% RSLogix 500 project PLC_Level_2_Project_9.RSS, saved by version 8.30.00.16 %
PROJECT "UNTITLED"    % processor: Bul.1763 MicroLogix 1100 Series B %

PROGRAM FILES
  LAD 2   8 rungs

DATA FILES
  O0 OUTPUT  4 elements
  I1 INPUT  6 elements
  S2 STATUS  66 elements
  B3 BINARY  1 elements
  T4 TIMER  1 elements
  C5 COUNTER  1 elements
  R6 CONTROL  1 elements
  N7 INTEGER  4 elements
  F8 FLOAT  1 elements
  ST9 STRING  8 elements

LADDER 2
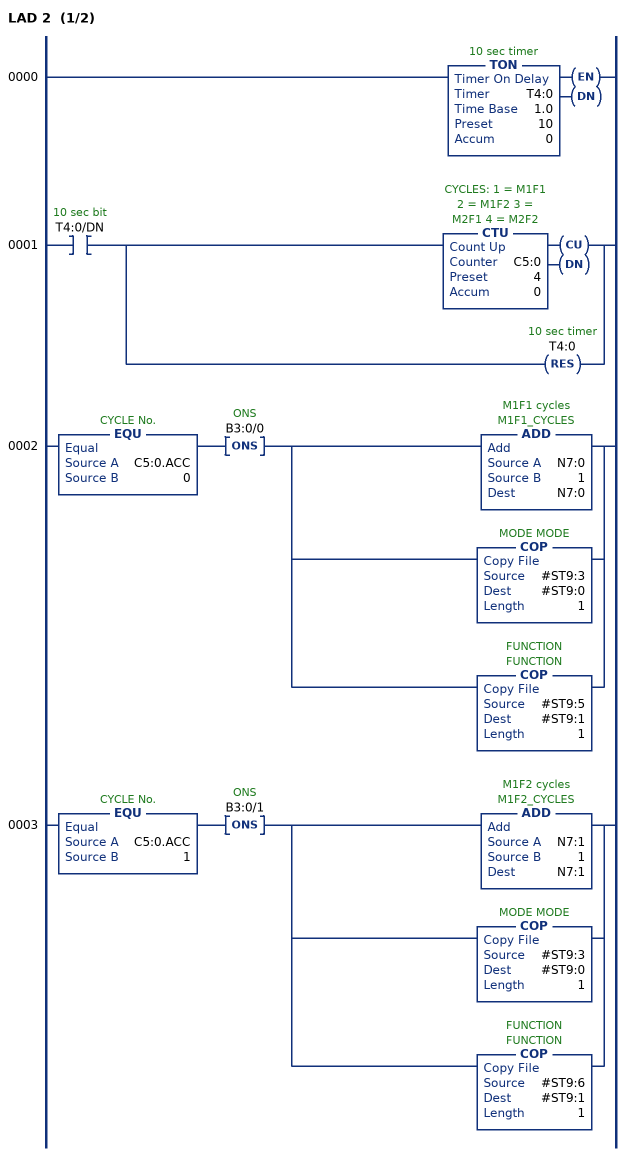
% Rung: 0 %
SOR TON T4:0 1.0 10 0 EOR
%   T4:0  "10 sec timer" %
% Rung: 1 %
SOR XIC T4:0/DN BST CTU C5:0 4 0 NXB RES T4:0 BND EOR
%   T4:0/DN  "10 sec bit" %
%   C5:0  "CYCLES: 1 = M1F1 2 = M1F2 3 = M2F1 4 = M2F2" %
%   T4:0  "10 sec timer" %
% Rung: 2 %
SOR EQU C5:0.ACC 0 ONS B3:0/0 BST ADD N7:0 1 N7:0 NXB COP #ST9:3 #ST9:0 1 NXB COP #ST9:5 #ST9:1 1 BND EOR
%   C5:0.ACC  "CYCLE No." %
%   B3:0/0  "ONS" %
%   N7:0  M1F1_CYCLES  "M1F1 cycles" %
%   ST9:3  "MODE-1" %
%   ST9:0  MODE  "MODE" %
%   ST9:5  "F1" %
%   ST9:1  FUNCTION  "FUNCTION" %
% Rung: 3 %
SOR EQU C5:0.ACC 1 ONS B3:0/1 BST ADD N7:1 1 N7:1 NXB COP #ST9:3 #ST9:0 1 NXB COP #ST9:6 #ST9:1 1 BND EOR
%   C5:0.ACC  "CYCLE No." %
%   B3:0/1  "ONS" %
%   N7:1  M1F2_CYCLES  "M1F2 cycles" %
%   ST9:3  "MODE-1" %
%   ST9:0  MODE  "MODE" %
%   ST9:6  "F2" %
%   ST9:1  FUNCTION  "FUNCTION" %

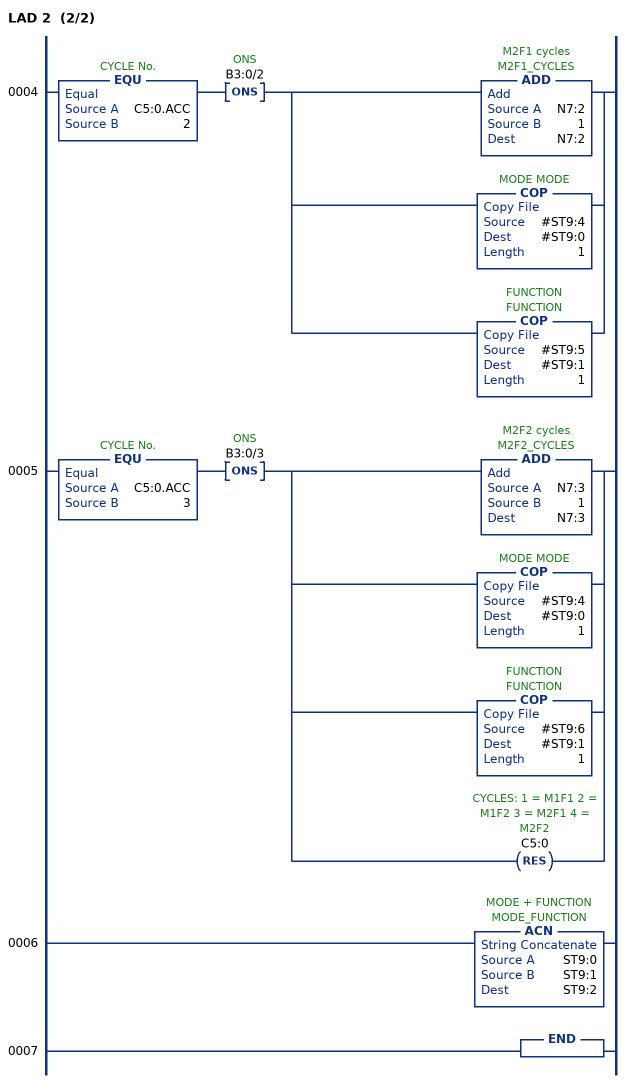
% Rung: 4 %
SOR EQU C5:0.ACC 2 ONS B3:0/2 BST ADD N7:2 1 N7:2 NXB COP #ST9:4 #ST9:0 1 NXB COP #ST9:5 #ST9:1 1 BND EOR
%   C5:0.ACC  "CYCLE No." %
%   B3:0/2  "ONS" %
%   N7:2  M2F1_CYCLES  "M2F1 cycles" %
%   ST9:4  "MODE-2" %
%   ST9:0  MODE  "MODE" %
%   ST9:5  "F1" %
%   ST9:1  FUNCTION  "FUNCTION" %
% Rung: 5 %
SOR EQU C5:0.ACC 3 ONS B3:0/3 BST ADD N7:3 1 N7:3 NXB COP #ST9:4 #ST9:0 1 NXB COP #ST9:6 #ST9:1 1 NXB RES C5:0 BND EOR
%   C5:0.ACC  "CYCLE No." %
%   B3:0/3  "ONS" %
%   N7:3  M2F2_CYCLES  "M2F2 cycles" %
%   ST9:4  "MODE-2" %
%   ST9:0  MODE  "MODE" %
%   ST9:6  "F2" %
%   ST9:1  FUNCTION  "FUNCTION" %
%   C5:0  "CYCLES: 1 = M1F1 2 = M1F2 3 = M2F1 4 = M2F2" %
% Rung: 6 %
SOR ACN ST9:0 ST9:1 ST9:2 EOR
%   ST9:0  MODE  "MODE" %
%   ST9:1  FUNCTION  "FUNCTION" %
%   ST9:2  MODE_FUNCTION  "MODE + FUNCTION" %
% Rung: 7 %
SOR END EOR

OTHER DOCUMENTED ADDRESSES
  B3:0/4  "REST VALUES"
  B3:0/5  "ONS"
  DFILE:0  "OUTPUT"
  DFILE:1  "INPUT"
  DFILE:2  "STATUS"
  DFILE:3  "BINARY"
  DFILE:4  "TIMER"
  DFILE:5  "COUNTER"
  DFILE:6  "CONTROL"
  DFILE:7  "INTEGER"
  DFILE:8  "FLOAT"
  DFILE:9  "STRING"
  ST9:7  "empty"
  ST9:7.0  "blank"

DATA TABLE (non-zero values as saved)
DATA T4
% .PRE .ACC %
% T4:0 % 10 0
DATA C5
% .PRE .ACC %
% C5:0 % 4 0
DATA ST9
% ST9:3 % "Mode-1"
% ST9:4 % "Mode-2"
% ST9:5 % "F1"
% ST9:6 % "F2"
